TYPE ST_SAFETY_FBMUTING:
STRUCT
	uStatus							: U_SAFETY_MUTING; 				(* Typ zalezny od bloku *)
	eState							: E_SAFETY_FBStateMUTING;		(* Enum ze statusem bloku *)
	bGeneralError					: BOOL; 						(* Gdy wystapi chociaz jeden Error *)
END_STRUCT
END_TYPE

(* stored: Version 1.1.0.1, ProductVersion 3.1.4022.12
   DUT ST_SAFETY_FBMUTING: Id {6d6c74c6-064b-4745-911d-15bb7f54c402} *)
